// SIMATIC S7-200 project (STEP 7-Micro/WIN), CPU 224 CN REL 02.02

ORGANIZATION_BLOCK 主程序:OB1
TITLE=程序注释
BEGIN
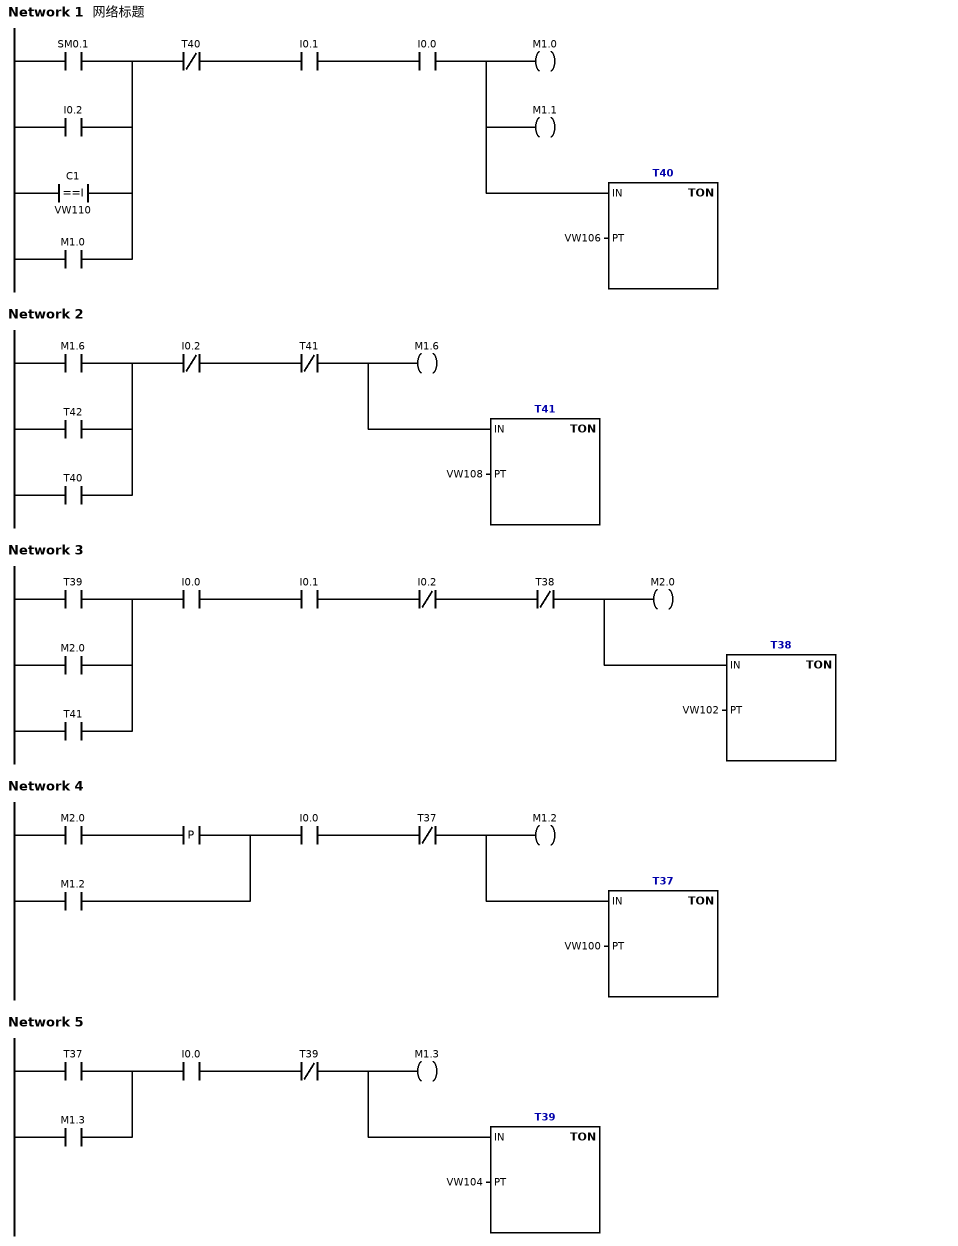
Network 1 // 网络标题
LD     SM0.1
O      I0.2
OW=    C1, VW110
O      M1.0
AN     T40
A      I0.1
A      I0.0
=      M1.0
=      M1.1
TON    T40, VW106
Network 2
LD     M1.6
O      T42
O      T40
AN     I0.2
AN     T41
=      M1.6
TON    T41, VW108
Network 3
LD     T39
O      M2.0
O      T41
A      I0.0
A      I0.1
AN     I0.2
AN     T38
=      M2.0
TON    T38, VW102
Network 4
LD     M2.0
EU
O      M1.2
A      I0.0
AN     T37
=      M1.2
TON    T37, VW100
Network 5
LD     T37
O      M1.3
A      I0.0
AN     T39
=      M1.3
TON    T39, VW104
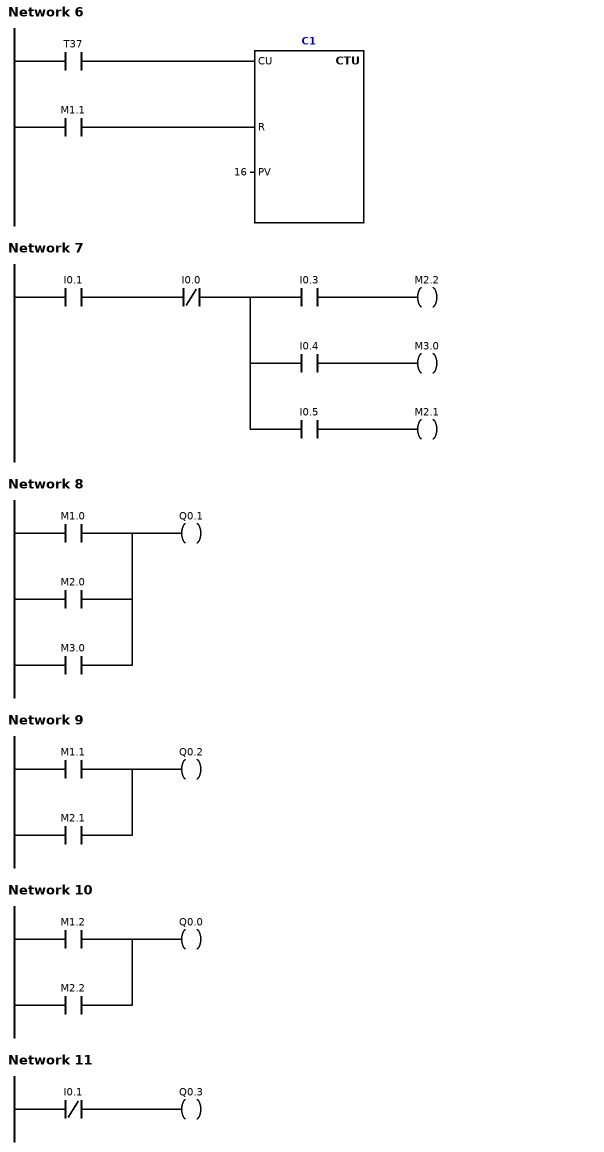
Network 6
LD     T37
LD     M1.1
CTU    C1, 16
Network 7
LD     I0.1
AN     I0.0
LPS
A      I0.3
=      M2.2
LRD
A      I0.4
=      M3.0
LPP
A      I0.5
=      M2.1
Network 8
LD     M1.0
O      M2.0
O      M3.0
=      Q0.1
Network 9
LD     M1.1
O      M2.1
=      Q0.2
Network 10
LD     M1.2
O      M2.2
=      Q0.0
Network 11
LDN    I0.1
=      Q0.3
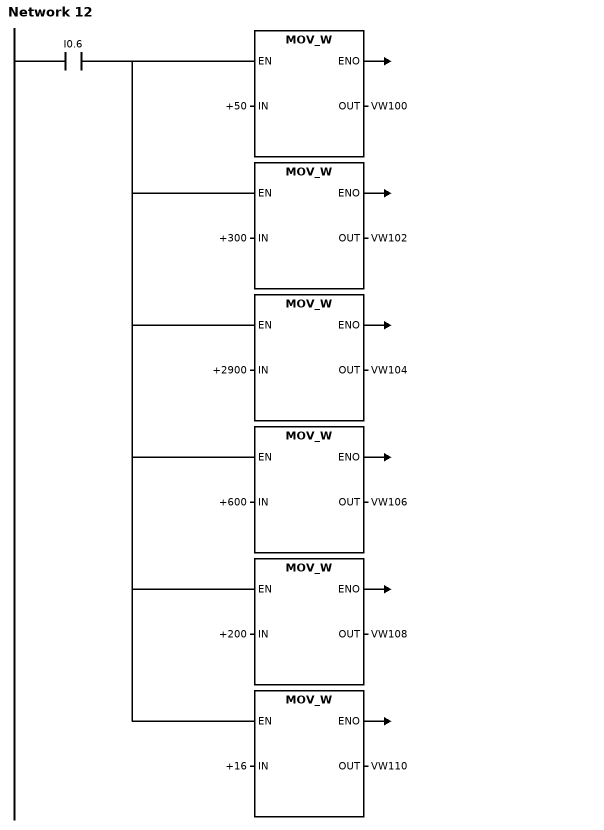
Network 12
LD     I0.6
MOVW   +50, VW100
MOVW   +300, VW102
MOVW   +2900, VW104
MOVW   +600, VW106
MOVW   +200, VW108
MOVW   +16, VW110
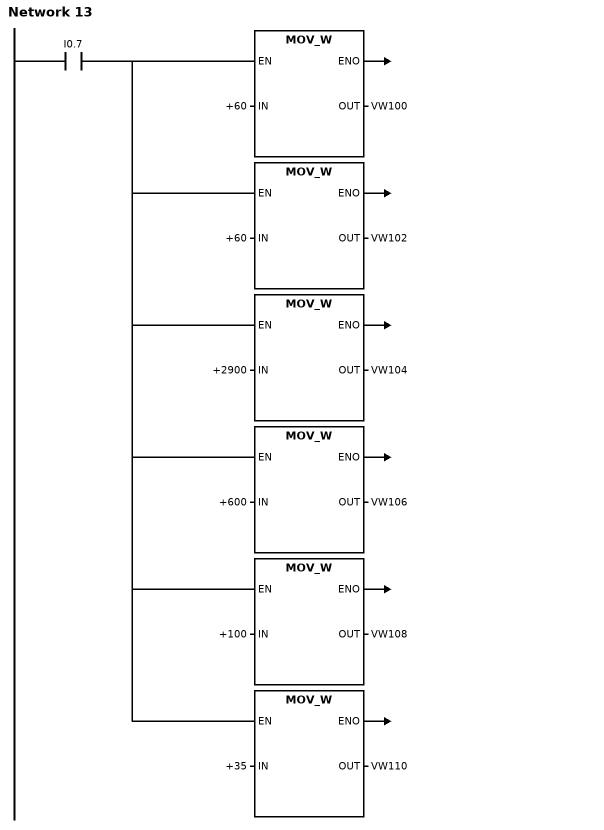
Network 13
LD     I0.7
MOVW   +60, VW100
MOVW   +60, VW102
MOVW   +2900, VW104
MOVW   +600, VW106
MOVW   +100, VW108
MOVW   +35, VW110
END_ORGANIZATION_BLOCK
